FUNCTION_BLOCK FB_Alarm IMPLEMENTS I_Alarm
VAR_INPUT
END_VAR
VAR_OUTPUT
END_VAR
VAR
	iAlarmNumber	:	UINT := 0;
	bTemporary		:	BOOL;
	bLatched		:	BOOL;
	sDescription	:	STRING;
	tsTimeOfOccur	:	TIMESTRUCT;
END_VAR

{attribute 'monitoring' := 'variable'}
PROPERTY AlarmNumber : UINT
GET
AlarmNumber := iAlarmNumber;
END_GET
SET
iAlarmNumber := AlarmNumber;
END_SET
END_PROPERTY

{attribute 'monitoring' := 'variable'}
PROPERTY Description : String
GET
Description := sDescription;
END_GET
SET
sDescription := Description;
END_SET
END_PROPERTY

METHOD Get : BOOL
VAR_INPUT
END_VAR
VAR_OUTPUT

END_VAR
Get := bLatched;
END_METHOD

METHOD Reset : BOOL
VAR_INPUT
END_VAR
IF NOT bTemporary THEN
	IF bLatched = TRUE THEN
		Reset := TRUE;
		bLatched := FALSE;
	END_IF
ELSE
	Reset := FALSE;
END_IF
END_METHOD

METHOD Set : BOOL
VAR
END_VAR
VAR_INPUT
	bIn	:	BOOL;
END_VAR
bTemporary := bIn;
IF NOT bLatched AND bIn THEN
	bLatched := TRUE;
	tsTimeOfOccur := GVL.fbMachineTime.systemTime;
END_IF
END_METHOD

PROPERTY TimeOfOccur : TIMESTRUCT
GET
TimeOfOccur := tsTimeOfOccur;
END_GET
END_PROPERTY

END_FUNCTION_BLOCK

(* stored: Version 1.1.0.1, ProductVersion 3.1.4024.12
   POU FB_Alarm: Id {bed2f1ec-601f-4cc2-8a29-1b808b16b28e}, SpecialFunc None
   Property AlarmNumber: Id {483a5e8f-e08f-4185-a7aa-e29351bf5027}
   Get Get: Id {209caddf-2723-419e-afb6-01275fd0d793}
   Set Set: Id {3cbb4afc-d1d2-491a-9f77-b34e764d4baa}
   Property Description: Id {214ab764-e938-4b63-851b-2218f8564a19}
   Get Get: Id {29352b5c-b26c-4cd7-a93f-441018d66c37}
   Set Set: Id {e64c5aac-4933-43de-a8dd-b3e48e9b6cb2}
   Method Get: Id {d062801b-a649-41fa-89db-fb1d0aae96e8}
   Method Reset: Id {de0d8ec5-fb9f-498f-bc79-30c4e4f55aa9}
   Method Set: Id {b7405dae-7583-4782-9136-6c5894abd4ae}
   Property TimeOfOccur: Id {c3b469ec-af3f-4075-a3f3-f61a65b94a03}
   Get Get: Id {23392ae3-de2a-4ecd-910f-83a62cf067a3} *)
